SUBAPPLICATION Uebung_011_AUDI (* Numeric Value Input *)
  (* Standard: 61499-2; Description: Copyright (c) 2023 Meisterschulen am Ostbahnhof This program and the accompanying materials are made available under the terms of the Eclipse Public License 2.0 which is available at https://www.eclipse.org/legal/epl-2.0/ SPDX-License-Identifier: EPL-2.0 *)
  (* Version 1.0, 2023-10-23, Franz Höpfinger, Meisterschulen am Ostbahnhof, initial API and implementation and/or initial documentation *)
  PACKAGE Uebungen;
  IMPORT Uebungen::const::UT::DefaultPool::InputNumber_I1;
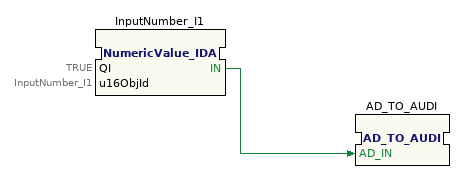
  FBS
    AD_TO_AUDI : adapter::conversion::unidirectional::AD_TO_AUDI;
    InputNumber_I1 : isobus::UT::io::NumericValue::NumericValue_IDA(QI := TRUE, u16ObjId := InputNumber_I1);
  END_FBS
  ADAPTER_CONNECTIONS
    InputNumber_I1.IN TO AD_TO_AUDI.AD_IN;
  END_CONNECTIONS
END_SUBAPPLICATION
